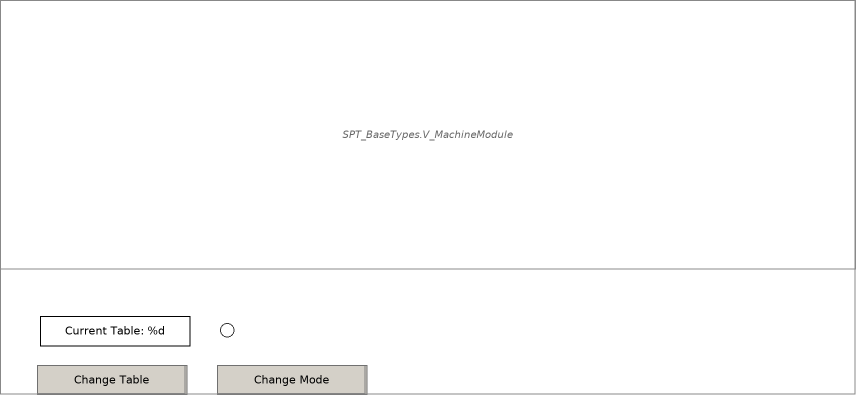
VISUALIZATION Visualization  // 856x395
    Frame (0,0 856x269)
        shows SPT_BaseTypes.V_MachineModule(HMI := MAIN.Machine.PackMLBaseModule_HMI)
    Button (37,365 150x30), "Change Table"
        toggle MAIN.Machine.CamModule.HMI.Cmd.ChangeTable
    Rectangle (40,316 150x30), "Current Table: %d", text variable: MAIN.Machine.CamModule.HMI.Sts.CurrentTable
    RadioButton (218,296 150x68), variable: MAIN.Machine.CamModule.HMI.Cfg.CamActivationMode
        Areas[0]: Text=Next Cycle
        Areas[1]: Text=As Soon As Possible
    Button (217,365 150x30), "Change Mode"
        toggle MAIN.Machine.CamModule.HMI.Cmd.ChangeMode
END_VISUALIZATION

(* stored: Version 1.1.0.1, ProductVersion 3.1.4024.12
   Visu Visualization: Id {dcda8cdc-31c0-441c-9c53-44fba7b7ab38} *)
